TYPE S_PT1T2_Param :
STRUCT
	K		: REAL;
	T1		: REAL;
	T2		: REAL;
END_STRUCT
END_TYPE

(* stored: Version 1.1.0.1, ProductVersion 3.1.4024.9
   DUT S_PT1T2_Param: Id {22fb11cc-28aa-4815-aa53-7d02370fd56e} *)
